# B&R Automation Studio project Pachore_Mayuresh_Project_1
Automation Studio 4.12.6.106; technology packages: Acp10Arnc0 5.24.1, mapp 5.24.1, mappView 5.24.4

## Configuration Config1

CPU X20CP1382, AutomationRuntime A4.83, Build 4.1.2, Safety 0.0, Vc V4.72.5

### Hardware
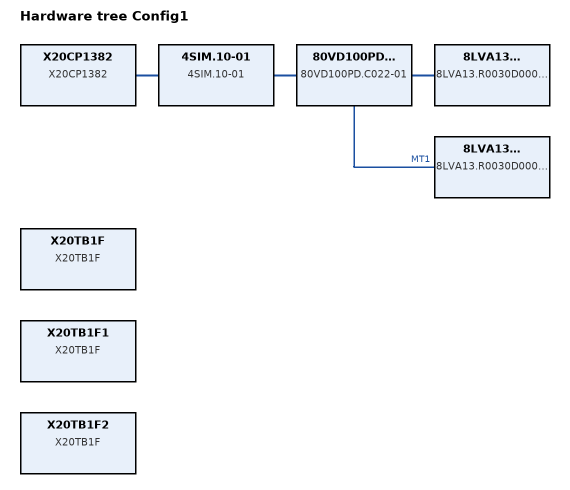
```
4SIM.10-01 : 4SIM.10-01 v1.3.0.0  [PLK1 -> X20CP1382.IF3 (NodeNumber=1) [Cable Type=PowerlinkCable, Length=10, Version=1.0.0.3]; PLK2 -> 80VD100PD.C022-01.PLK1 (NodeNumber=1) [Cable Type=PowerlinkCable, Length=10, Version=1.0.0.3]]
  Supervision = off
80VD100PD.C022-01 : 80VD100PD.C022-01 v2.5.0.0  [PLK1 -> 4SIM.10-01.PLK2 (NodeNumber=2) [Cable Type=PowerlinkCable, Length=10, Version=1.0.0.3]; MT2 -> 8LVA13.R0030D000-0.MT]
  MotionTP = Acp10Arnc0
  AxisIsPeriodic_r1 = on
  Period_r1 = 360
  BothEndSwitchesAreNormallyOpen_r1 = on
  QuickStopIsNormallyOpen_r1 = on
  AxisIsPeriodic_r2 = on
  Period_r2 = 360
  BothEndSwitchesAreNormallyOpen_r2 = on
  QuickStopIsNormallyOpen_r2 = on
8LVA13.R0030D000-0 : 8LVA13.R0030D000-0 v2.2.0.4  [MT -> 80VD100PD.C022-01.MT2]
8LVA13.R0030D000-0a : 8LVA13.R0030D000-0 v2.2.0.4  [MT -> 80VD100PD.C022-01.MT1]
X20CP1382 : X20CP1382 v1.14.0.0  [X1 -> X1.SL; X2 -> X2.SL; X3 -> X3.SL]
  Module X1 (Type=X1, Virtual=true, Version=1.14.0.0)
    Connection (Connector=SS1, TargetModule=X20TB1F, TargetConnector=SS)
    Connection (Connector=SL, TargetModule=X20CP1382, TargetConnector=X1)
  Module X2 (Type=X2, Virtual=true, Version=1.14.0.0)
    Connection (Connector=SS1, TargetModule=X20TB1F1, TargetConnector=SS)
    Connection (Connector=SL, TargetModule=X20CP1382, TargetConnector=X2)
  Module X3 (Type=X3, Virtual=true, Version=1.14.0.0)
    Connection (Connector=SS1, TargetModule=X20TB1F2, TargetConnector=SS)
    Connection (Connector=SL, TargetModule=X20CP1382, TargetConnector=X3)
  Connector IF2:
    ActivateDevice = 1
    Mode = Manual
    InternetAddress = 192.168.0.1
    SubnetMask = 255.255.255.0
    ActivateSnmp = 2
  Connector IF3:
    CycleTime = 2000
  ConfigurationID = UniboTest2024_Config1
  TimerDeviceType = EPLX2X
  TimerDevice = X20CP1382.IF3
  TaskClassIdleTime = 6000
  Cyclic1Duration = 2000
  Cyclic1Tolerance = 0
  ActivateOpcUa = 1
  OpcUaInformationModels_PV_Version = 1
X20TB1F : X20TB1F v1.0.0.0
X20TB1F1 : X20TB1F v1.0.0.0
X20TB1F2 : X20TB1F v1.0.0.0
```

### IoMap.iom - X20CP1382/IoMap.iom
```iecst
VAR_CONFIG
	::Conv_Lock AT %IX."4SIM.10-01".DigitalInput01;
	::Cutter_Lock AT %IX."4SIM.10-01".DigitalInput02;
	::Start_Button AT %IX."4SIM.10-01".DigitalInput03;
	::Stop_Button AT %IX."4SIM.10-01".DigitalInput04;
	::Sensor_Button AT %IX."4SIM.10-01".DigitalInput05;
	::Reset_Button AT %IX."4SIM.10-01".DigitalInput06;
	::Speed AT %IW."4SIM.10-01".AnalogInput01;
	::Position AT %IW."4SIM.10-01".AnalogInput02;
	::DI1.LED_Light AT %QX."4SIM.10-01".DigitalOutput01;
	::DI2.LED_Light AT %QX."4SIM.10-01".DigitalOutput02;
	::DI3.LED_Light AT %QX."4SIM.10-01".DigitalOutput05;
	::DI4.LED_Light AT %QX."4SIM.10-01".DigitalOutput06;
	::DI5.LED_Light AT %QX."4SIM.10-01".DigitalOutput10;
	::DI6.LED_Light AT %QX."4SIM.10-01".DigitalOutput12;
	::Display AT %QW."4SIM.10-01".AnalogOutput01;
END_VAR
```

### Acp10cfg.ncc - X20CP1382/Motion/Acp10cfg.ncc
```
NcConfiguration (Version=5.20.1, NcSwId=Acp10)
  ACP10CF1_typ:
    cnt_nettrc_rec_drive = 150
    bufsize_trace_upload = 1200
    tc_nc_man_task = Cyclic #1
    glob_pv_as_ncobject = Yes
    ncsys_dl_broadcast = Yes
    ncsys_dl_acp_reset = Yes
    safemc_log_err_to_ax = Yes
    network_init:
      ncsw_init_execute = Yes
      automatic_execute = No
      node_nr_warning = Yes
      net_err_before_ncact = Yes
    nettrc:
      enter_parsecrec = Yes
      enter_ncaction = Yes
      save_ring_startidx = No
    cam_prof_download:
      cam_dat_dl_parallel = No
      tc_cam_dl_parallel = Task class for NC Manager task
    plk_if[0]:
      if_name = IF3
      tc_CycDat_PLCopen = Task class for NC Manager task
      mc_broadcast_extdat = No
```

### Config.mpaxisbasic - X20CP1382/Motion/Config.mpaxisbasic
```
Element gAxisBasic_Master (Type=mpaxisbasic)
Element gAxisBasic_Slave (Type=mpaxisbasic)
```

## Logical view

Binary libraries used (declarations not repeated): operator, runtime, astime, AsIecCon, sys_lib, brsystem, Acp10man, Acp10par, NcGlobal, Acp10sim, Acp10_MC, MpAxis, AsTCP, standard, AsArLog, AsBrStr, MpBase, MpCom, AsIODiag

### MNG_Package.var
```iecst
(*                                                                            *)
(* File generated by the B&R AS 4 control config generator                    *)
(*                                                                            *)
(*     Provider: machineering                                                 *)
(*  Application: industrialPhysics_2.4.master                                 *)
(* Architecture: Windows 64 Bit                                               *)
(*      Version: 2.4.10491.master                                             *)
(*        Build: 164f85bec                                                    *)
(*         Date: 2020-03-30, Time: 13:49:25                                   *)
(*                                                                            *)

                VAR
                ComTCP_SimInputs : ComTCP_INPUTS_32BIT := (0);
    ComTCP_SimOutputs : ComTCP_OUTPUTS_32BIT := (0);

    ComTCP_SimServerAddress : STRING[15] := '127.0.0.1';
    ComTCP_SimServerPort : UINT := 5000;
    ComTCP_SimSendCycleTime : TIME := T#10ms;
    ComTCP_SimActive : BOOL := FALSE;

                END_VAR
```

### MNG_Package.typ
```iecst
(*                                                                            *)
(* File generated by the B&R AS 4 control config generator                    *)
(*                                                                            *)
(*     Provider: machineering                                                 *)
(*  Application: industrialPhysics_2.4.master                                 *)
(* Architecture: Windows 64 Bit                                               *)
(*      Version: 2.4.10491.master                                             *)
(*        Build: 164f85bec                                                    *)
(*         Date: 2020-03-30, Time: 13:49:25                                   *)
(*                                                                            *)

TYPE
ComTCP_INPUTS_32BIT : STRUCT

		NumSignals	: INT := 15;

        Emergency_Button_ButtonToggle : BOOL := 0;
        (* BOOL Emergency_Button_ButtonToggle *)
        Yellow_Button_ButtonPress : BOOL := 0;
        (* BOOL Yellow_Button_ButtonPress *)
        White_Button_ButtonPress : BOOL := 0;
        (* BOOL White_Button_ButtonPress *)
        Start_Button_ButtonPress : BOOL := 0;
        (* BOOL Start_Button_ButtonPress *)
        Stop_Button_ButtonPress : BOOL := 0;
        (* BOOL Stop_Button_ButtonPress *)
        Knob_0_AXIS : REAL := 0.0;
        (* REAL Knob_0_AXIS *)
        Knob_1_AXIS : REAL := 0.0;
        (* REAL Knob_1_AXIS *)
        Knob_2_AXIS : REAL := 0.0;
        (* REAL Knob_2_AXIS *)
        Knob_3_AXIS : REAL := 0.0;
        (* REAL Knob_3_AXIS *)
        Shaft_1_AXIS : REAL := 0.0;
        (* REAL Shaft_1_AXIS *)
        Shaft_1_LBK : BOOL := 0;
        (* BOOL Shaft_1_LBK *)
        Shaft_1_LFR : BOOL := 0;
        (* BOOL Shaft_1_LFR *)
        Shaft_0_AXIS : REAL := 0.0;
        (* REAL Shaft_0_AXIS *)
        Shaft_0_LBK : BOOL := 0;
        (* BOOL Shaft_0_LBK *)
        Shaft_0_LFR : BOOL := 0;
        (* BOOL Shaft_0_LFR *)

	END_STRUCT;

ComTCP_OUTPUTS_32BIT : STRUCT

		NumSignals	: INT := 6;

        Yellow_light_Key : UDINT := 0;
        (* UDINT Yellow_light_Key *)
        Stop_light_Key : UDINT := 0;
        (* UDINT Stop_light_Key *)
        White_light_Key : UDINT := 0;
        (* UDINT White_light_Key *)
        Green_light_Key : UDINT := 0;
        (* UDINT Green_light_Key *)
        Shaft_0_ACT_POS : REAL := 0.0;
        (* REAL Shaft_0_ACT_POS *)
        Shaft_1_ACT_POS : REAL := 0.0;
        (* REAL Shaft_1_ACT_POS *)

	END_STRUCT;

END_TYPE
```

### Global.var - Global variables
```iecst
(*Name of Axis*)
VAR
	gAxis01 : ACP10AXIS_typ;
	gAxis02 : ACP10AXIS_typ;
END_VAR
(*Hardware Variables*)
VAR
	Conv_Lock : BOOL;
	Cutter_Lock : BOOL;
	Start_Button : BOOL;
	Stop_Button : BOOL;
	Sensor_Button : BOOL;
	Reset_Button : BOOL;
	Speed : INT;
	Position : INT;
	DI1 : FSM_LED;
	DI2 : FSM_LED;
	DI3 : FSM_LED;
	DI4 : FSM_LED;
	DI5 : FSM_LED;
	DI6 : FSM_LED;
	Display : INT;
END_VAR
(*HMI Variables*)
VAR
	Emergancy_Button_HMI : BOOL;
	Start_Button_HMI : BOOL;
	Stop_Button_HMI : BOOL;
	Sensor_Button_HMI : BOOL;
	Reset_Button_HMI : BOOL;
	Conv_Lock_HMI : BOOL;
	Cutter_Lock_HMI : BOOL;
	Conv_Speed_HMI : REAL;
	Cutter_Speed_HMI : REAL;
	Cutting_Pos_HMI : REAL;
	Cutting_Depth_HMI : REAL;
	Blade_Man_HMI : REAL;
	Conv_Man_HMI : REAL;
	Slow_Blade_HMI : BOOL;
	Slow_Conv_HMI : BOOL;
	LED_DI1_HMI : BOOL;
	LED_DI2_HMI : BOOL;
	LED_DI3_HMI : BOOL;
	LED_DI4_HMI : BOOL;
	LED_DI5_HMI : BOOL;
	LED_DI6_HMI : BOOL;
	Dis_Conv_Speed_HMI : REAL;
	Dis_Cut_Speed_HMI : REAL;
	Dis_Cut_Pos_HMI : INT;
	Dis_Cut_Depth_HMI : INT;
	Man_Mode_HMI : BOOL;
	Over_Ride_HMI : BOOL;
END_VAR
(*LED_IO Variables*)
VAR
	Power_Axis : BOOL;
	Home_Axis : BOOL;
	Reset_Command : BOOL;
	Error_Command : BOOL;
	Start_Command : BOOL := FALSE;
	Stop_Command : BOOL := TRUE;
END_VAR
(*Master Variables*)
VAR
	Master : FSM_AXIS;
	M_Active : BOOL;
	M_Actual_Position : REAL;
	M_Actual_Velocity : REAL;
	M_Homed : BOOL;
	M_Powered : BOOL;
	M_Stoped : BOOL;
	Do_Cut : BOOL := FALSE;
	Done_Cut : BOOL := FALSE;
END_VAR
(*Slave Variables*)
VAR
	Slave : FSM_AXIS;
	S_Active : BOOL;
	S_Actual_Position : REAL;
	S_Actual_Velocity : REAL;
	S_Homed : BOOL;
	S_Powered : BOOL;
	S_Stoped : BOOL;
END_VAR
(*Input Bridge Variables*)
VAR
	Start_Trigger : BOOL;
	Stop_Trigger : BOOL;
	Error_Trigger : BOOL;
	Reset_Trigger : BOOL;
	Sensor_Trigger : BOOL;
	Conv_Lock_HMI_Trigger : BOOL;
	Conv_Lock_Trigger : BOOL;
	Cutter_Lock_HMI_Trigger : BOOL;
	Cutter_Lock_Trigger : BOOL;
	Slow_Blade_Trigger : BOOL;
	Slow_Conv_Trigger : BOOL;
	Over_Ride_Trigger : BOOL;
	Conv_Speed : REAL;
	Cut_Pos : REAL;
	Cutter_Speed : REAL;
	Cut_depth : REAL;
	Blade_Pos : REAL;
	Conv_Pos : REAL;
	M_Error : BOOL;
	S_Error : BOOL;
END_VAR
(*Manual Motion Variables*)
VAR
	Manual_Mode_Trigger : BOOL;
	Man_Mode_OFF : BOOL := TRUE;
END_VAR
```

### Package Logical/Libraries - Global libraries

### Library Logical/Libraries/ComTCP/ComTCP_L (ANSIC)

#### MNG_ComHdlr.cpp
```cpp
#include "MNG_ComHdlr.hpp"
#include "MNG_CpyMsgToInp.cpp"
#include "MNG_CpyOutToMsg.cpp"

asTcpFcn_t _asTcpFcn;

MNG_ComHdlr::MNG_ComHdlr(char *srvIpAdr, unsigned int srvPort, TIME sendCycleTime)
{
	_srvIpAdr = srvIpAdr;
	_srvPort = srvPort;
	_sendCycleTime = sendCycleTime;
	InitParams();
}

MNG_ComHdlr::~MNG_ComHdlr()
{
}

int MNG_ComHdlr::RunCommunication(void* pSimInputs, void* pSimOutputs, BOOL* pSimActive) {

        unsigned long int _lastCounter = _counter;

	ComTCP_INPUTS_32BIT_FWRD* pFwrd_SimInputs = static_cast<ComTCP_INPUTS_32BIT_FWRD*>((pSimInputs));
	ComTCP_OUTPUTS_32BIT_FWRD* pFwrd_SimOutputs = static_cast<ComTCP_OUTPUTS_32BIT_FWRD*>((pSimOutputs));

	switch (_internalState) {

		case MNG_Init:
                        *pSimActive = FALSE;
			_asTcpFcn.tcpOpen.enable = FALSE;
			TcpOpen(&_asTcpFcn.tcpOpen);
			_asTcpFcn.tcpIoctl.enable = FALSE;
			TcpIoctl(&_asTcpFcn.tcpIoctl);
			_asTcpFcn.tcpClient.enable = FALSE;
			TcpClient(&_asTcpFcn.tcpClient);
			_asTcpFcn.tcpSend.enable = FALSE;
			TcpSend(&_asTcpFcn.tcpSend);
			_asTcpFcn.tcpRecv.enable = FALSE;
			TcpRecv(&_asTcpFcn.tcpRecv);
			_asTcpFcn.tcpClose.enable = FALSE;
			TcpClose(&_asTcpFcn.tcpClose);

			_connectionTon.IN = FALSE;
			_connectionTon.PT = _connectionTime;
			_sendTon.IN = FALSE;
			_sendTon.PT = _sendCycleTime;
			SetStateValue(MNG_Socket);
			break;

		case MNG_Socket:
                        *pSimActive = FALSE;
			init_TcpSocket();
			TcpOpen(&_asTcpFcn.tcpOpen);
			_recvOffset = 0;
			if (_connect == 1) {
				SetStateValue(MNG_Open);
				_connectionTon.IN = FALSE;
			}
			break;

		case MNG_Open:
                        *pSimActive = FALSE;
			init_TcpOpen();
			TcpOpen(&_asTcpFcn.tcpOpen);
			if (_asTcpFcn.tcpOpen.status == 0) {
				SetStateValue(MNG_SetIo);
				_asTcpFcn.tcpIoctl.enable = FALSE;
				TcpIoctl(&_asTcpFcn.tcpIoctl);
				_connectionTon.IN = FALSE;
			}
			break;

		case MNG_SetIo:
                        *pSimActive = FALSE;
			init_TcpIoctl();
			TcpIoctl(&_asTcpFcn.tcpIoctl);
			if (_asTcpFcn.tcpIoctl.status == 0) {
				SetStateValue(MNG_Linger);
				_asTcpFcn.tcpClient.enable = FALSE;
				TcpClient(&_asTcpFcn.tcpClient);
				_connectionTon.IN = FALSE;
			}
			break;

		case MNG_Linger:
                        *pSimActive = FALSE;
			init_TcpLinger();
			TcpIoctl(&_asTcpFcn.tcpIoctl);

			if (_asTcpFcn.tcpIoctl.status == 0) {
				SetStateValue(MNG_Connecting);
				_asTcpFcn.tcpClient.enable = FALSE;
				_connectionTon.IN = FALSE;
			}

		case MNG_Connecting:
                        *pSimActive = FALSE;
			_asTcpFcn.tcpClient.enable = TRUE;
			_asTcpFcn.tcpClient.ident = _asTcpFcn.tcpOpen.ident;
			_asTcpFcn.tcpClient.portserv = _srvPort;
			_asTcpFcn.tcpClient.pServer = (long)_srvIpAdr;
			TcpClient(&_asTcpFcn.tcpClient);

			if (_asTcpFcn.tcpClient.status == ERR_FUB_BUSY) {
				// state = state || SetStateValue(Connecting);
			} else if (_asTcpFcn.tcpClient.status == 0) {
				SetStateValue(MNG_Exchange);
				_connectionTon.IN = FALSE;
				SetSendDone(TRUE);
			}
			break;

		case MNG_Exchange:
			init_TcpRecv();
			TcpRecv(&_asTcpFcn.tcpRecv);

			if (_asTcpFcn.tcpRecv.status==0){
                        *pSimActive = FALSE;
			_connectionTon.IN = FALSE;
			_recvLen = _asTcpFcn.tcpRecv.recvlen;
			_potMsgLen = N_TO_HUDINT(_recvBuffer[3]) + SIXTEEN;
			_totalRecvLen = _recvOffset + _recvLen;

			if ((_totalRecvLen < SIXTEEN) || (_totalRecvLen < _potMsgLen)) {
			_recvOffset = _recvOffset + _recvLen;
			}	else {
			while ((_potMsgLen > 0) && (_potMsgLen <= _totalRecvLen)) {
			// misconfigured message sizes
                        if ((unsigned long int)_potMsgLen > sizeof(_recvMessage)) {
			SetStateValue(MNG_Reset);
			break;
			}

			brsmemcpy((unsigned long int) &_recvMessage, (unsigned long int) &_recvBuffer, _potMsgLen*sizeof(unsigned long int));
			_totalRecvLen = _totalRecvLen - _potMsgLen;
			brsmemmove((unsigned long int) &_recvBuffer, (unsigned long int) &_recvBuffer + _potMsgLen, _totalRecvLen*sizeof(unsigned long int));
			_counter = MNG_CpyMsgToInp(&_recvMessage,pFwrd_SimInputs);
                        *pSimActive = (_lastCounter != _counter);
			_recvOffset = _totalRecvLen;

			if (_totalRecvLen > SIXTEEN) {
			_potMsgLen = N_TO_HUDINT(_recvBuffer[3]) + SIXTEEN;
			} else {
			_potMsgLen = 0;
			}

			}
			}
			}

			_sendTon.IN = _sendDone;
			TON(&_sendTon);

			if (_sendTon.Q || _asTcpFcn.tcpSend.enable == 1) {
				if (_sendDone==TRUE) {
					SetSendDone(FALSE);
					MNG_CpyOutToMsg(&_sendMessage, _counter,pFwrd_SimOutputs);
					init_TcpSend(pFwrd_SimOutputs);
				}
				TcpSend(&_asTcpFcn.tcpSend);

				if (_asTcpFcn.tcpSend.status == 0) {
					if (_asTcpFcn.tcpSend.datalen != _asTcpFcn.tcpSend.sentlen) {
						// state = state || SetStateValue(Exchange);
					}
					_asTcpFcn.tcpSend.enable = FALSE;
					SetSendDone(TRUE);
				}
			}
			if (_asTcpFcn.tcpRecv.status == tcpERR_NOT_CONNECTED) {
				SetStateValue(MNG_Closing);
			}
			break;

		case MNG_Closing:
                        *pSimActive = FALSE;
			_asTcpFcn.tcpClose.enable = TRUE;
			_asTcpFcn.tcpClose.ident = _asTcpFcn.tcpOpen.ident;
			_asTcpFcn.tcpClose.how = 0;
			TcpClose(&_asTcpFcn.tcpClose);

			if(_asTcpFcn.tcpClose.status == 0 || _asTcpFcn.tcpClose.status == 32600){
				SetStateValue(MNG_Init);
			}
			break;

                case MNG_Reset:
                        SetStateValue(MNG_Closing);
                        break;
	}

	TON(&_connectionTon);
	_connectionTon.IN = TRUE;
	if (_connectionTon.Q == 1) {
		SetStateValue(MNG_Closing);
		_connectionTon.IN = FALSE;
	}

	return _internalState;
}

void MNG_ComHdlr::init_TcpOpen(){
	_asTcpFcn.tcpOpen.enable = _connect;
}

void MNG_ComHdlr::init_TcpSocket(){
	_asTcpFcn.tcpOpen.enable = TRUE;
	_asTcpFcn.tcpOpen.pIfAddr = 0;
	_asTcpFcn.tcpOpen.port = PORT;
	_asTcpFcn.tcpOpen.options = tcpOPT_REUSEADDR;
}

void MNG_ComHdlr::init_TcpIoctl(){
	_asTcpFcn.tcpIoctl.enable = TRUE;
	_asTcpFcn.tcpIoctl.pData = (unsigned long int) &_one;
	_asTcpFcn.tcpIoctl.datalen = 4;
	_asTcpFcn.tcpIoctl.ident = _asTcpFcn.tcpOpen.ident;
	_asTcpFcn.tcpIoctl.ioctl = tcpTCP_NODELAY_SET;
}

void MNG_ComHdlr::init_TcpLinger(){
	_asTcpFcn.tcpLINGER.lLinger = FALSE;
	_asTcpFcn.tcpLINGER.lOnOff = TRUE;
	_asTcpFcn.tcpIoctl.enable = TRUE;
	_asTcpFcn.tcpIoctl.pData = (unsigned long int) &_asTcpFcn.tcpLINGER;
	_asTcpFcn.tcpIoctl.datalen = sizeof(_asTcpFcn.tcpLINGER);
	_asTcpFcn.tcpIoctl.ident = _asTcpFcn.tcpOpen.ident;
	_asTcpFcn.tcpIoctl.ioctl = tcpSO_LINGER_SET;
}

void MNG_ComHdlr::init_TcpClient(){

	_asTcpFcn.tcpClient.enable = TRUE;
	_asTcpFcn.tcpClient.ident = _asTcpFcn.tcpOpen.ident;
	_asTcpFcn.tcpClient.portserv = _srvPort;
	_asTcpFcn.tcpClient.pServer = (long)_srvIpAdr;
}

void MNG_ComHdlr::init_TcpRecv(){

	_asTcpFcn.tcpRecv.enable = TRUE;
	_asTcpFcn.tcpRecv.ident= _asTcpFcn.tcpOpen.ident;
	_asTcpFcn.tcpRecv.datamax = sizeof(_recvBuffer) - _recvOffset;
	_asTcpFcn.tcpRecv.pData = (unsigned long int) &_recvBuffer + _recvOffset;
}

void MNG_ComHdlr::init_TcpSend(ComTCP_OUTPUTS_32BIT_FWRD *pSimOutputs){

	_asTcpFcn.tcpSend.enable = TRUE;
	_asTcpFcn.tcpSend.ident= _asTcpFcn.tcpOpen.ident;
	_asTcpFcn.tcpSend.datalen = 16 + ((pSimOutputs->NumSignals) + 1) * 4;
	_asTcpFcn.tcpSend.pData = (unsigned long int)&_sendMessage;
	_asTcpFcn.tcpSend.flags = 0;
}

void MNG_ComHdlr::InitParams(){
	_internalState = MNG_Init;
	_connectionTime = 3000;
	_one=1;
	_connect = TRUE;
	_potMsgLen = 0;
	_recvLen = 0;
	_recvOffset = 0;
	_counter = 0;
	SetSendDone(FALSE);
}

void MNG_ComHdlr::SetSendDone(bool toggle){
	_sendDone=toggle;
}

void MNG_ComHdlr::SetStateValue(MNG_internalState_t stateVal){
	_internalState=stateVal;
}
```

#### MNG_CpyOutToMsg.cpp
```cpp
#include "MNG_InternalTyp.hpp"

unsigned long int MNG_CpyOutToMsg(MNG_RawDatagram * pToServer, unsigned long int counter, ComTCP_OUTPUTS_32BIT_FWRD *pSimOutputs ) {

        unsigned long int DWordBuffer;

        pSimOutputs->NumSignals = 6;
        (pToServer->Header).ByteCount    = H_TO_NUDINT(28);
        (pToServer->Header).DatagramType = H_TO_NUDINT(MNG_Raw32BitImage);
        (pToServer->Header).SentTime = H_TO_NUDINT(0);  // Todo
        (pToServer->Header).Counter = H_TO_NUDINT(counter);
        pToServer->Payload[0] = H_TO_NUDINT(pSimOutputs->NumSignals);

    /* Yellow_light_Key : UINT32 */
    pToServer->Payload[1] = H_TO_NUDINT(pSimOutputs->Yellow_light_Key);

    /* Stop_light_Key : UINT32 */
    pToServer->Payload[2] = H_TO_NUDINT(pSimOutputs->Stop_light_Key);

    /* White_light_Key : UINT32 */
    pToServer->Payload[3] = H_TO_NUDINT(pSimOutputs->White_light_Key);

    /* Green_light_Key : UINT32 */
    pToServer->Payload[4] = H_TO_NUDINT(pSimOutputs->Green_light_Key);

    /* Shaft_0_ACT_POS : FLOAT32 */
    brsmemcpy((unsigned long int)&(DWordBuffer), (unsigned long int)&(pSimOutputs->Shaft_0_ACT_POS), 4);
    pToServer->Payload[5] = H_TO_NUDINT(DWordBuffer);

    /* Shaft_1_ACT_POS : FLOAT32 */
    brsmemcpy((unsigned long int)&(DWordBuffer), (unsigned long int)&(pSimOutputs->Shaft_1_ACT_POS), 4);
    pToServer->Payload[6] = H_TO_NUDINT(DWordBuffer);

	return 0;
}
```

### Library Logical/Libraries/My_Library (IEC)

#### FSM_AXIS.st
```iecst
FUNCTION_BLOCK FSM_AXIS

	CASE State OF
		0://Initiation
			Power_ON := FALSE;

			IF RS_Valid AND RS_Disabled THEN
				State 	:= 2;
				Active 	:= TRUE;
			END_IF

			IF RS_Errorstop AND RS_Valid THEN
				State 	:= 1;
			END_IF

		1://Error
			V_Execute 	:= FALSE;
			Add_Execute := FALSE;
			A_Execute 	:= FALSE;

			IF Reset_Error THEN
				R_Execute := TRUE;
				IF R_Done AND P_Status THEN
					State := 3;
				END_IF
				IF R_Done AND NOT P_Status THEN
					State := 2;
				END_IF
			END_IF

		2://Disabled
			P_Enable := FALSE;
			Power_ON := FALSE;

			IF Error THEN
				State := 1;
			ELSIF Home THEN
				State := 4;
			ELSIF Power THEN
				State := 3;
			END_IF

		3://StandStill

			P_Enable := TRUE;
			Power_ON := TRUE;

			IF Error THEN
				State 			:= 1;
			ELSIF Home AND NOT Is_Homed THEN
				State 			:= 4;
			ELSIF NOT Power THEN
				State 			:= 2;
			ELSIF Move_Velocity THEN
				Move_Abs_Done 	:= FALSE;
				Move_Add_Done 	:= FALSE;
				Stop_Done 		:= FALSE;
				State 			:= 5;
			ELSIF Move_Additive AND NOT Move_Additive_Old THEN
				Move_Abs_Done 	:= FALSE;
				Move_Add_Done 	:= FALSE;
				Stop_Done 		:= FALSE;
				State 			:= 6;
			ELSIF Move_Absolute AND NOT Move_Absolute_Old THEN
				Move_Abs_Done 	:= FALSE;
				Move_Add_Done 	:= FALSE;
				Stop_Done 		:= FALSE;
				State 			:= 7;
			ELSIF Stop THEN
				State 			:= 8;
			END_IF

		4://Homing Axis

			H_Execute := TRUE;
			IF Error THEN
				State 		:= 1;
				H_Execute 	:= FALSE;
			ELSIF H_Done AND Power THEN
				State 		:= 3;
				H_Execute 	:= FALSE;
				Is_Homed 	:= TRUE;
			ELSIF H_Done AND NOT Power THEN
				State 		:= 2;
				H_Execute 	:= FALSE;
				Is_Homed 	:= TRUE;
			END_IF

		5://Moving Axis in Velocity mode

			P_Enable 	:= TRUE;
			V_Execute 	:= TRUE;
			IF Old_Velocity <> Velocity THEN
				V_Execute := FALSE;
			END_IF

			IF Error THEN
				State := 1;
			ELSIF Move_Additive THEN
				State := 6;
			ELSIF Move_Absolute THEN
				State := 7;
			ELSIF NOT Power OR Stop THEN
				State := 8;
			END_IF

		6://Moving Axis in Additive mode

			P_Enable 	:= TRUE;
			Add_Execute := TRUE;

			IF Error THEN
				State 			:= 1;
			END_IF
			IF NOT Power OR Stop THEN
				State 			:= 8;
				Add_Execute 	:= FALSE;
			END_IF
			IF Add_Done THEN
				Move_Add_Done 	:= TRUE;
				Add_Execute 	:= FALSE;
				State 			:= 3;
			END_IF

		7://Moving Axis in Absolute Mode

			P_Enable 	:= TRUE;
			A_Execute 	:= TRUE;

			IF Error THEN
				State 			:= 1;
			END_IF
			IF NOT Power OR Stop THEN
				State 			:= 8;
				A_Execute 		:= FALSE;
			END_IF
			IF A_Done THEN
				Move_Abs_Done 	:= TRUE;
				A_Execute 		:= FALSE;
				State 			:= 3;
			END_IF

		8://Stopping Axis

			P_Enable 	:= TRUE;
			S_Execute 	:= TRUE;

			IF Error THEN
				State 		:= 1;
			END_IF
			IF S_Done THEN
				V_Execute 	:= FALSE;
				S_Execute 	:= FALSE;
				Stop_Done 	:= TRUE;
				State 		:= 3;
			END_IF
			IF RS_Errorstop AND RS_Valid THEN
				S_Execute 	:= FALSE;
				State 		:= 1;
			END_IF

	END_CASE

	Move_Absolute_Old 		:= Move_Absolute;
	Move_Additive_Old 		:= Move_Additive;
	Old_Velocity 			:= Velocity;

	//Calling all PLCopen function blocks used
	//Read Status
	MCRS(	Axis 			:= Axis_Name,
			Enable 			:= TRUE);
	RS_Valid 				:= MCRS.Valid;
	RS_Error 				:= MCRS.Error;
	RS_Errorstop 			:= MCRS.Errorstop;
	RS_Disabled 			:= MCRS.Disabled;
	//Power
	MCP(	Axis 			:= Axis_Name,
			Enable 			:= P_Enable);
	P_Status 				:= MCP.Status;
	P_Error 				:= MCP.Error;
	//Home
	MCH(	Axis 			:= Axis_Name,
			Execute 		:= H_Execute);
	H_Done 					:= MCH.Done;
	H_Error					:= MCH.Error;
	//Stop
	MCS(	Axis 			:= Axis_Name,
			Execute 		:= S_Execute,
			Deceleration 	:= Deceleration);
	S_Done 					:= MCS.Done;
	S_Error 				:= MCS.Error;
	//Reset
	MCR(	Axis 			:= Axis_Name,
			Execute			:= R_Execute);
	R_Done 					:= MCR.Done;
	R_Error 				:= MCR.Error;
	//Read Actual Position
	MCRAP(	Axis 			:= Axis_Name,
			Enable 			:= TRUE);
	RAP_Valid 				:= MCRAP.Valid;
	RAP_Error 				:= MCRAP.Error;
	Actual_Position 		:= MCRAP.Position;
	//Read Actual Velocity
	MCRAV(	Axis 			:= Axis_Name,
			Enable 			:= TRUE);
	RAV_Valid 				:= MCRAV.Valid;
	RAV_Error 				:= MCRAV.Error;
	Actual_Velocity 		:= MCRAV.Velocity;
	//Move Velocity
	MCMV(	Axis 			:= Axis_Name,
			Execute 		:= V_Execute,
			Velocity 		:= Velocity,
			Acceleration 	:= Acceleration,
			Deceleration 	:= Deceleration,
			Direction 		:= Direction);
	V_Error 				:= MCMV.Error;
	//Move Additive
	MCMAdd(	Axis 			:= Axis_Name,
			Execute 		:= Add_Execute,
			Distance 		:= Distance,
			Velocity 		:= Velocity,
			Acceleration 	:= Acceleration,
			Deceleration 	:= Deceleration);
	Add_Done 				:= MCMAdd.Done;
	Add_Error 				:= MCMAdd.Error;
	//Move Absolute
	MCMA(	Axis 			:= Axis_Name,
			Execute 		:= A_Execute,
			Position 		:= Position,
			Velocity 		:= Velocity,
			Acceleration 	:= Acceleration,
			Deceleration 	:= Deceleration,
			Direction 		:= Direction);
	A_Done 					:= MCMA.Done;
	A_Error 				:= MCMA.Error;

	Error := RS_Error OR P_Error OR H_Error OR S_Error OR R_Error OR RAP_Error OR RAV_Error OR V_Error OR Add_Error OR A_Error;

END_FUNCTION_BLOCK
```

#### FSM_LED.st
```iecst
(* For Turning LED ON/OFF/Blink *)
FUNCTION_BLOCK FSM_LED

	IF LED_State = 'on' THEN
		LED_Light := TRUE;
	END_IF

	IF LED_State = 'off' THEN
		LED_Light := FALSE;
	END_IF

	IF LED_State = 'blink' THEN

		CASE State OF

			0:
				Timer(IN := TRUE, PT := T#500ms);
				IF Timer.Q = TRUE THEN
					Timer(IN 	:= FALSE);
					LED_Light 	:= TRUE;
					State 		:= 1;
				END_IF

			1:
				Timer(IN := TRUE, PT := T#500ms);
				IF Timer.Q = TRUE THEN
					Timer(IN 	:= FALSE);
					LED_Light 	:= FALSE;
					State 		:= 0;
				END_IF
		END_CASE

	END_IF

END_FUNCTION_BLOCK
```


- Data object Logical/gAxis01obj/gAxis01i (Ax) (no source held here)

- Data object Logical/gAxis02obj/gAxis02i (Ax) (no source held here)

### Data object Logical/MyCam (Cam)

- Visualisation Logical/mappView (not shown)

### Program Logical/Master (IEC)

#### Variables.var
```iecst
VAR
	M_Move_Velocity : BOOL;
	M_Move_Additive : BOOL;
	M_Move_Absolute : BOOL;
	M_Stop : BOOL;
	State : INT := 0;
	M_Position : REAL;
	one_time : BOOL;
	M_Move_Additive_Done : BOOL;
	M_Move_Absolute_Done : BOOL;
	M_Distance : REAL;
	M_Direction : USINT := 0;
	M_Velocity : REAL;
END_VAR
```

#### Main.st
```iecst
PROGRAM _INIT
	(* Insert code here *)

END_PROGRAM

PROGRAM _CYCLIC

	CASE State OF
		0://Initialization

			IF M_Active AND M_Homed AND M_Powered THEN
				State := 2;
			END_IF
			IF Manual_Mode_Trigger THEN
				State := 5;
			END_IF

		1://Error and Stopping

			M_Move_Velocity := FALSE;
			M_Move_Additive := FALSE;
			M_Move_Absolute := FALSE;
			M_Stop 			:= TRUE;

			IF M_Stoped THEN
				M_Move_Velocity := FALSE;
				M_Move_Additive := FALSE;
				M_Move_Absolute := FALSE;
				M_Stop 			:= FALSE;
				State 			:= 2;
			END_IF

		2://Standstill

			IF NOT Error_Command AND Start_Command AND Man_Mode_OFF AND (NOT Do_Cut OR Done_Cut) THEN
				State := 3;
			END_IF
			IF Manual_Mode_Trigger THEN
				State := 5;
			END_IF

		3://Moving Conveyor
			M_Velocity 		:= Conv_Speed;
			M_Move_Velocity := TRUE;
			M_Move_Additive := FALSE;
			M_Move_Absolute := FALSE;
			M_Stop 			:= FALSE;

			Do_Cut 		:= FALSE;
			Done_Cut 	:= FALSE;

			IF Stop_Command OR Error_Command THEN
				State := 1;
			ELSIF Sensor_Trigger THEN
				State := 4;
			ELSIF Manual_Mode_Trigger THEN
				State := 5;
			END_IF

		4://Reaching Cutting Position
			M_Distance 		:= Cut_Pos;
			M_Velocity 		:= Conv_Speed;
			M_Move_Velocity := FALSE;
			M_Move_Additive := TRUE;
			M_Move_Absolute := FALSE;
			M_Stop 			:= FALSE;

			IF M_Move_Additive_Done THEN
				State 			:= 1;
				Do_Cut 			:= TRUE;
				M_Move_Velocity := FALSE;
				M_Move_Additive := FALSE;
				M_Move_Absolute := FALSE;
				M_Stop 			:= FALSE;
				one_time 		:= FALSE;
			END_IF

			IF Stop_Command OR Error_Command THEN
				State := 1;
			END_IF

			IF Done_Cut AND NOT (Stop_Command OR Error_Command) THEN
				State := 2;
			END_IF

			IF Manual_Mode_Trigger THEN
				State := 5;
			END_IF

		5://Running in Manual Mode
			Power_Axis 		:= TRUE;
			Man_Mode_OFF 	:= FALSE;
			M_Move_Velocity := TRUE;
			M_Move_Additive := FALSE;
			M_Move_Absolute := FALSE;
			M_Stop 			:= FALSE;

			M_Velocity 		:= Conv_Pos;
			M_Direction 	:= 0;
			IF M_Velocity < 0 THEN
				M_Velocity 	:= -Conv_Pos;
				M_Direction := 1;
			END_IF
			IF NOT Manual_Mode_Trigger THEN
				Power_Axis 		:= FALSE;
				Start_Command 	:= FALSE;
				M_Move_Velocity := FALSE;
				M_Move_Additive := FALSE;
				M_Move_Absolute := FALSE;
				M_Stop 			:= FALSE;
				State 			:= 2;
			END_IF

			IF Error_Command THEN
				State := 1;
			END_IF

	END_CASE

	//Calling FSM_AXIS Function
	Master(	Axis_Name 		:= ADR(gAxis01),
			Acceleration 	:= 5000,
			Deceleration 	:= 5000,
			Position 		:= M_Position,
			Distance 		:= M_Distance,
			Velocity 		:= M_Velocity,
			Direction 		:= M_Direction,
			Home 			:= Home_Axis,
			Power 			:= Power_Axis,
			Move_Velocity 	:= M_Move_Velocity,
			Move_Absolute 	:= M_Move_Absolute,
			Move_Additive 	:= M_Move_Additive,
			Stop 			:= M_Stop,
			Reset_Error 	:= Reset_Command);
	M_Active 				:= Master.Active;
	M_Actual_Position		:= Master.Actual_Position;
	M_Actual_Velocity 		:= Master.Actual_Velocity;
	M_Move_Absolute_Done 	:= Master.Move_Abs_Done;
	M_Move_Additive_Done 	:= Master.Move_Add_Done;
	M_Homed 				:= Master.Is_Homed;
	M_Powered 				:= Master.Power_ON;
	M_Stoped 				:= Master.Stop_Done;
	M_Error 				:= Master.Error;

END_PROGRAM

PROGRAM _EXIT
	(* Insert code here *)

END_PROGRAM
```

### Program Logical/Slave (IEC)

#### Variables.var
```iecst
VAR
	State : INT := 0;
	S_Move_Velocity : BOOL;
	S_Move_Absolute : BOOL;
	S_Move_Additive : BOOL;
	S_Stop : BOOL;
	S_Move_Absolute_Done : BOOL;
	S_Direction : USINT;
	S_Move_Additive_Done : BOOL;
	S_Position : REAL;
	S_Distance : REAL;
	S_Velocity : REAL;
END_VAR
```

#### Main.st
```iecst
PROGRAM _INIT
	(* Insert code here *)

END_PROGRAM

PROGRAM _CYCLIC

	CASE State OF
		0://Initiation

			Done_Cut 	:= FALSE;
			Do_Cut 		:= FALSE;
			State 		:= 1;

		1://Standstill

			IF NOT Error_Command AND Start_Command AND Do_Cut AND Man_Mode_OFF THEN
				S_Velocity 	:= Cutter_Speed;
				State 		:= 2;     //Uncomment for Cutter in Cam similar Mechanism
				//State 		:= 4;   //Uncomment for Cutter in Lead Screw Mechanism
			END_IF

			IF Manual_Mode_Trigger THEN
				State := 6;
			END_IF

		2://Cutting Considering it as a Cam cutter
			S_Move_Velocity := FALSE;
			S_Move_Absolute := TRUE;
			S_Move_Additive := FALSE;
			S_Stop 			:= FALSE;
			S_Position 		:= Cut_depth;
			S_Direction 	:= 0;

			IF S_Actual_Position = 0.0 THEN
				S_Move_Absolute_Done := FALSE;
			END_IF

			IF S_Move_Absolute_Done THEN
				State 			:= 3;
				S_Move_Velocity := FALSE;
				S_Move_Absolute := FALSE;
				S_Move_Additive := FALSE;
				S_Stop 			:= FALSE;
			END_IF

			IF Stop_Command OR Error_Command OR NOT Do_Cut THEN
				State 			:= 1;
				S_Move_Velocity := FALSE;
				S_Move_Absolute := FALSE;
				S_Move_Additive := FALSE;
				S_Stop 			:= FALSE;
			END_IF

		3://Retracting Considering it as a Cam cutter
			S_Move_Velocity := FALSE;
			S_Move_Absolute := TRUE;
			S_Move_Additive := FALSE;
			S_Stop 			:= FALSE;
			S_Position 		:= 0.0;
			S_Direction 	:= 1;

			IF S_Actual_Position <> 0.0 THEN
				S_Move_Absolute_Done := FALSE;
			END_IF

			IF S_Move_Absolute_Done THEN
				State 			:= 1;
				Do_Cut 			:= FALSE;
				Done_Cut 		:= TRUE;
				S_Move_Velocity := FALSE;
				S_Move_Absolute := FALSE;
				S_Move_Additive := FALSE;
				S_Stop 			:= FALSE;
			END_IF

			IF Stop_Command OR Error_Command OR NOT Do_Cut THEN
				State 			:= 1;
				S_Move_Velocity := FALSE;
				S_Move_Absolute := FALSE;
				S_Move_Additive := FALSE;
				S_Stop 			:= FALSE;
			END_IF

		4://Cutting Considering a lead Screw Cutter
			S_Move_Velocity := FALSE;
			S_Move_Absolute := FALSE;
			S_Move_Additive := TRUE;
			S_Stop 			:= FALSE;
			S_Distance 		:= Cut_depth;

			IF S_Actual_Position = 0.0 THEN
				S_Move_Additive_Done := FALSE;
			END_IF

			IF S_Move_Additive_Done THEN
				State 			:= 5;
				S_Move_Velocity := FALSE;
				S_Move_Absolute := FALSE;
				S_Move_Additive := FALSE;
				S_Stop 			:= FALSE;
			END_IF

			IF Stop_Command OR Error_Command OR NOT Do_Cut THEN
				State 			:= 1;
				S_Move_Velocity := FALSE;
				S_Move_Absolute := FALSE;
				S_Move_Additive := FALSE;
				S_Stop 			:= FALSE;
			END_IF

		5://Retracting Considering a lead Screw Cutter
			S_Move_Velocity := FALSE;
			S_Move_Absolute := FALSE;
			S_Move_Additive := TRUE;
			S_Stop 			:= FALSE;
			S_Distance 		:= -Cut_depth;

			IF S_Actual_Position <> 0.0 THEN
				S_Move_Additive_Done := FALSE;
			END_IF

			IF S_Move_Additive_Done THEN
				State 			:= 1;
				Do_Cut 			:= FALSE;
				Done_Cut 		:= TRUE;
				S_Move_Velocity := FALSE;
				S_Move_Absolute := FALSE;
				S_Move_Additive := FALSE;
				S_Stop 			:= FALSE;
			END_IF

			IF Stop_Command OR Error_Command OR NOT Do_Cut THEN
				State 			:= 1;
				S_Move_Velocity := FALSE;
				S_Move_Absolute := FALSE;
				S_Move_Additive := FALSE;
				S_Stop 			:= FALSE;
			END_IF

		6: //Running in Manual Mode
			Power_Axis 		:= TRUE;
			Man_Mode_OFF 	:= FALSE;
			S_Move_Velocity := TRUE;
			S_Move_Additive := FALSE;
			S_Move_Absolute := FALSE;
			S_Stop 			:= FALSE;

			S_Velocity 		:= Blade_Pos;
			S_Direction 	:= 0;

			IF S_Velocity < 0 THEN
				S_Velocity 	:= -Blade_Pos;
				S_Direction := 1;
			END_IF
			IF Error_Command THEN
				State := 1;
			END_IF

			IF NOT Manual_Mode_Trigger THEN
				S_Move_Absolute_Done 	:= FALSE;
				State 					:= 7;
			END_IF

		7: //Sending Cutter Back to Original Position
			IF S_Actual_Position <> 0.0 THEN
				S_Velocity 		:= 50;
				S_Move_Velocity := FALSE;
				S_Move_Absolute := TRUE;
				S_Move_Additive := FALSE;
				S_Stop 			:= FALSE;
				S_Position 		:= 0.0;
				S_Direction 	:= 1;

				IF Error_Command THEN
					State := 1;
				END_IF
			END_IF
			IF S_Actual_Position = 0.0 THEN
				Man_Mode_OFF 	:= TRUE;
				State 			:= 1;
				Power_Axis 		:= FALSE;
				S_Move_Velocity := FALSE;
				S_Move_Absolute := FALSE;
				S_Move_Additive := FALSE;
				S_Stop 			:= FALSE;
			END_IF

			IF Error_Command THEN
				State := 1;
			END_IF

	END_CASE

	//Calling FSM_AXIS Function
	Slave(	Axis_Name 		:= ADR(gAxis02),
			Acceleration 	:= 5000,
			Deceleration 	:= 5000,
			Position 		:= S_Position,
			Distance 		:= S_Distance,
			Velocity 		:= S_Velocity,
			Direction 		:= S_Direction,
			Home 			:= Home_Axis,
			Power 			:= Power_Axis,
			Move_Velocity 	:= S_Move_Velocity,
			Move_Absolute 	:= S_Move_Absolute,
			Move_Additive 	:= S_Move_Additive,
			Stop 			:= S_Stop,
			Reset_Error 	:= Reset_Command);
	S_Active 				:= Slave.Active;
	S_Actual_Position 		:= Slave.Actual_Position;
	IF State = 3 OR State = 5 THEN
		S_Actual_Velocity := -Slave.Actual_Velocity;
	ELSE
		S_Actual_Velocity := Slave.Actual_Velocity;
	END_IF

	S_Move_Absolute_Done 	:= Slave.Move_Abs_Done;
	S_Move_Additive_Done 	:= Slave.Move_Add_Done;
	S_Homed 				:= Slave.Is_Homed;
	S_Powered 				:= Slave.Power_ON;
	S_Stoped 				:= Slave.Stop_Done;
	S_Error 				:= Slave.Error;

END_PROGRAM

PROGRAM _EXIT
	(* Insert code here *)

END_PROGRAM
```

### Program Logical/LED_IO (IEC)

#### Variables.var
```iecst
VAR
	State : INT := 0;
END_VAR
```

#### Main.st
```iecst
PROGRAM _INIT
	(* Insert code here *)

END_PROGRAM

PROGRAM _CYCLIC
	(* Insert code here *)
	(* Insert code here *)
	CASE State OF
		0: //Initiation
			DI1(LED_State := 'off');
			DI2(LED_State := 'off');
			DI3(LED_State := 'off');
			DI4(LED_State := 'off');
			DI5(LED_State := 'off');
			DI6(LED_State := 'off');

			IF M_Active AND Man_Mode_OFF THEN
				State := 2;
			END_IF

		1: //Error

			DI1(LED_State := 'off');
			DI2(LED_State := 'off');
			DI3(LED_State := 'off');
			DI4(LED_State := 'off');
			DI5(LED_State := 'off');
			DI6(LED_State := 'blink');

			Error_Command 	:= TRUE;
			Start_Command 	:= FALSE;
			Stop_Command 	:= TRUE;
			Power_Axis 		:= FALSE;

			IF Reset_Trigger AND Error_Trigger THEN
				Reset_Command 	:= TRUE;
				Error_Command 	:= FALSE;
			ELSIF Reset_Trigger AND NOT Error_Trigger THEN
				Reset_Command 	:= FALSE;
				Error_Command 	:= FALSE;
				State 			:= 2;
			END_IF

		2: //Disabled

			IF Error_Trigger THEN
				State 		:= 1;
			ELSIF Reset_Trigger THEN
				Power_Axis 	:= TRUE;
			END_IF

			DI1(LED_State := 'on');
			DI2(LED_State := 'on');
			DI3(LED_State := 'on');
			DI4(LED_State := 'on');
			DI5(LED_State := 'on');
			DI6(LED_State := 'on');

			IF M_Powered AND M_Homed THEN
				State := 4;
			ELSIF M_Powered AND NOT M_Homed THEN
				State := 3;
			END_IF
			IF NOT Man_Mode_OFF THEN
				State := 0;
			END_IF

		3: //Homing
			DI1(LED_State := 'blink');
			DI2(LED_State := 'blink');
			DI3(LED_State := 'blink');
			DI4(LED_State := 'blink');
			DI5(LED_State := 'blink');
			DI6(LED_State := 'blink');

			Home_Axis := TRUE;

			IF Error_Trigger THEN
				State 		:= 1;
			ELSIF M_Homed THEN
				Home_Axis 	:= FALSE;
				State 		:= 4;
			END_IF

			IF NOT Man_Mode_OFF THEN
				State := 0;
			END_IF

		4://Ready
			IF NOT (Conv_Lock_Trigger OR Conv_Lock_HMI_Trigger) THEN
				DI1(LED_State := 'off');
			END_IF
			IF NOT (Cutter_Lock_Trigger OR Cutter_Lock_HMI_Trigger) THEN
				DI2(LED_State := 'off');
			END_IF
			IF (Conv_Lock_Trigger OR Conv_Lock_HMI_Trigger) THEN
				DI1(LED_State := 'on');
			END_IF
			IF (Cutter_Lock_Trigger OR Cutter_Lock_HMI_Trigger) THEN
				DI2(LED_State := 'on');
			END_IF

			DI3(LED_State := 'blink');
			DI4(LED_State := 'off');
			DI5(LED_State := 'off');
			DI6(LED_State := 'off');

			Power_Axis := TRUE;

			IF Error_Trigger THEN
				State := 1;
			ELSIF Start_Trigger AND NOT Error_Trigger THEN
				State := 5;
			END_IF
			IF NOT Man_Mode_OFF THEN
				State := 0;
			END_IF

		5://Run
			IF NOT (Conv_Lock_Trigger OR Conv_Lock_HMI_Trigger) THEN
				DI1(LED_State := 'off');
			END_IF
			IF NOT (Cutter_Lock_Trigger OR Cutter_Lock_HMI_Trigger) THEN
				DI2(LED_State := 'off');
			END_IF
			IF (Conv_Lock_Trigger OR Conv_Lock_HMI_Trigger) THEN
				DI1(LED_State := 'on');
			END_IF
			IF (Cutter_Lock_Trigger OR Cutter_Lock_HMI_Trigger) THEN
				DI2(LED_State := 'on');
			END_IF

			DI3(LED_State := 'on');
			DI4(LED_State := 'on');
			DI5(LED_State := 'off');
			DI6(LED_State := 'off');

			Start_Command 	:= TRUE;
			Stop_Command 	:= FALSE;

			IF Error_Trigger THEN
				State := 1;
			ELSIF Sensor_Trigger THEN
				State := 8;
			ELSIF Stop_Trigger THEN
				Stop_Command 	:= TRUE;
				State 			:= 10;
			END_IF
			IF NOT Man_Mode_OFF THEN
				State := 0;
			END_IF

		8://Sensor Triggered
			IF NOT (Conv_Lock_Trigger OR Conv_Lock_HMI_Trigger) THEN
				DI1(LED_State := 'off');
			END_IF
			IF NOT (Cutter_Lock_Trigger OR Cutter_Lock_HMI_Trigger) THEN
				DI2(LED_State := 'off');
			END_IF
			IF (Conv_Lock_Trigger OR Conv_Lock_HMI_Trigger) THEN
				DI1(LED_State := 'on');
			END_IF
			IF (Cutter_Lock_Trigger OR Cutter_Lock_HMI_Trigger) THEN
				DI2(LED_State := 'on');
			END_IF

			DI3(LED_State := 'on');
			DI4(LED_State := 'on');
			DI5(LED_State := 'on');
			DI6(LED_State := 'off');

			IF Do_Cut THEN
				State := 9;
			ELSIF Stop_Trigger THEN
				Stop_Command 	:= TRUE;
				State 			:= 10;
			END_IF

			IF Error_Trigger THEN
				State := 1;
			END_IF

		9://Cutting in Operation
			IF NOT (Conv_Lock_Trigger OR Conv_Lock_HMI_Trigger) THEN
				DI1(LED_State := 'off');
			END_IF
			IF NOT (Cutter_Lock_Trigger OR Cutter_Lock_HMI_Trigger) THEN
				DI2(LED_State := 'off');
			END_IF
			IF (Conv_Lock_Trigger OR Conv_Lock_HMI_Trigger) THEN
				DI1(LED_State := 'on');
			END_IF
			IF (Cutter_Lock_Trigger OR Cutter_Lock_HMI_Trigger) THEN
				DI2(LED_State := 'on');
			END_IF

			DI3(LED_State := 'on');
			DI4(LED_State := 'on');
			DI5(LED_State := 'blink');
			DI6(LED_State := 'off');

			IF Done_Cut THEN
				State := 5;
			ELSIF Stop_Trigger THEN
				Stop_Command 	:= TRUE;
				State 			:= 10;
			END_IF

			IF Error_Trigger THEN
				State := 1;
			END_IF

		10://Stop

			Start_Command := FALSE;

			IF Error_Trigger THEN
				State := 1;
			ELSIF M_Stoped THEN
				State := 4;
			END_IF
			IF NOT Man_Mode_OFF THEN
				State := 0;
			END_IF

	END_CASE

END_PROGRAM

PROGRAM _EXIT
	(* Insert code here *)

END_PROGRAM
```

### Program Logical/Input_Bridge (IEC)

#### Main.st
```iecst
PROGRAM _INIT
	(* Insert code here *)
	//Initial Parameters

	Conv_Speed 		:= 100;
	Cut_Pos 		:= 50;
	Cutter_Speed 	:= 20;
	Cut_depth 		:= 50;

END_PROGRAM

PROGRAM _CYCLIC

	IF DiagCpuIsSimulated() THEN
		(* For Simulation *)
		//Operator
		//LED_IO Bridge
		Start_Trigger 			:= ComTCP_SimInputs.Start_Button_ButtonPress 		OR Start_Button_HMI;
		Stop_Trigger 			:= ComTCP_SimInputs.Stop_Button_ButtonPress 		OR Stop_Button_HMI;
		Error_Trigger 			:= ComTCP_SimInputs.Emergency_Button_ButtonToggle 	OR Emergancy_Button_HMI OR M_Error OR S_Error;
		Reset_Trigger 			:= ComTCP_SimInputs.White_Button_ButtonPress 		OR Reset_Button_HMI;
		Sensor_Trigger 			:= ComTCP_SimInputs.Yellow_Button_ButtonPress 		OR Sensor_Button_HMI;
		Conv_Lock_HMI_Trigger 	:= Conv_Lock_HMI;
		Cutter_Lock_HMI_Trigger := Cutter_Lock_HMI;

		IF Conv_Lock_HMI_Trigger THEN
			IF Conv_Speed_HMI < 10 THEN
				Conv_Speed 	:= 10;
			ELSE
				Conv_Speed 	:= Conv_Speed_HMI;
			END_IF
			IF Cutting_Pos_HMI < 10 THEN
				Cut_Pos 	:= 10;
			ELSE
				Cut_Pos 	:= Cutting_Pos_HMI;
			END_IF
		END_IF

		IF Cutter_Lock_HMI_Trigger THEN
			IF Cutter_Speed_HMI < 10 THEN
				Cutter_Speed 	:= 10;
			ELSE
				Cutter_Speed 	:= Cutter_Speed_HMI;
			END_IF
			IF Cutting_Depth_HMI < 10 THEN
				Cut_depth 		:= 10;
			ELSE
				Cut_depth 		:= Cutting_Depth_HMI;
			END_IF
		END_IF

		//Manual Motion
		Manual_Mode_Trigger := Man_Mode_HMI;
		Slow_Blade_Trigger 	:= Slow_Blade_HMI;
		Slow_Conv_Trigger 	:= Slow_Conv_HMI;
		IF Slow_Blade_Trigger THEN
			Blade_Pos := Blade_Man_HMI * 0.01 * 1000;
		ELSE
			Blade_Pos := Blade_Man_HMI * 1000;
		END_IF

		IF Slow_Conv_Trigger THEN
			Conv_Pos := Conv_Man_HMI * 0.01 *1000;
		ELSE
			Conv_Pos := Conv_Man_HMI * 1000;
		END_IF

	ELSE
		(* For Actual Setup *)
		Start_Trigger 			:= Start_Button OR Start_Button_HMI;
		Stop_Trigger 			:= Stop_Button OR Stop_Button_HMI;
		Error_Trigger 			:= Emergancy_Button_HMI OR M_Error OR S_Error;
		Reset_Trigger 			:= Reset_Button OR Reset_Button_HMI;
		Sensor_Trigger 			:= Sensor_Button OR Sensor_Button_HMI;
		Conv_Lock_HMI_Trigger 	:= Conv_Lock_HMI;
		Cutter_Lock_HMI_Trigger := Cutter_Lock_HMI;
		Conv_Lock_Trigger 		:= Conv_Lock;
		Cutter_Lock_Trigger 	:= Cutter_Lock;
		Over_Ride_Trigger 		:= Over_Ride_HMI;
		IF Over_Ride_Trigger THEN
			IF Conv_Lock_HMI_Trigger THEN
				IF Conv_Speed_HMI < 10 THEN
					Conv_Speed 	:= 10;
				ELSE
					Conv_Speed 	:= Conv_Speed_HMI;
				END_IF
				IF Cutting_Pos_HMI < 10 THEN
					Cut_Pos 	:= 10;
				ELSE
					Cut_Pos 	:= Cutting_Pos_HMI;
				END_IF
			END_IF
			IF Cutter_Lock_HMI_Trigger THEN
				IF Cutter_Speed_HMI < 10 THEN
					Cutter_Speed 	:= 10;
				ELSE
					Cutter_Speed 	:= Cutter_Speed_HMI;
				END_IF
				IF Cutting_Depth_HMI < 10 THEN
					Cut_depth 		:= 10;
				ELSE
					Cut_depth 		:= Cutting_Depth_HMI;
				END_IF
			END_IF
		ELSE
			IF Conv_Lock_Trigger AND NOT Cutter_Lock_Trigger THEN
				Conv_Speed 			:= (Speed*3000/32767);
				IF Speed < 10 THEN
					Conv_Speed 		:= 10;
				END_IF
				Cut_Pos 			:= (Position*1000/32767);
				IF Position < 10 THEN
					Cut_Pos 		:= 10;
				END_IF

			ELSIF Cutter_Lock_Trigger AND NOT Conv_Lock_Trigger THEN
				Cutter_Speed 		:= (Speed*3000/32767);
				IF Speed < 10 THEN
					Cutter_Speed 	:= 10;
				END_IF
				Cut_depth 			:= (Position*360/32767);
				IF Position < 10 THEN
					Cut_depth 		:= 10;
				END_IF
			ELSIF Conv_Lock_Trigger AND Cutter_Lock_Trigger THEN
				Error_Trigger 	:= TRUE;
			END_IF
		END_IF

		//Manual Motion
		Manual_Mode_Trigger := Man_Mode_HMI;
		Slow_Blade_Trigger 	:= Slow_Blade_HMI;
		Slow_Conv_Trigger 	:= Slow_Conv_HMI;
		IF Slow_Blade_Trigger THEN
			Blade_Pos 	:= Blade_Man_HMI * 0.01 * 1000;
		ELSE
			Blade_Pos 	:= Blade_Man_HMI*1000;
		END_IF

		IF Slow_Conv_Trigger THEN
			Conv_Pos 	:= Conv_Man_HMI * 0.01 * 1000;
		ELSE
			Conv_Pos 	:= Conv_Man_HMI*1000;
		END_IF
	END_IF

END_PROGRAM

PROGRAM _EXIT
	(* Insert code here *)

END_PROGRAM
```

### Program Logical/Output_Bridge (IEC)

#### Main.st
```iecst
PROGRAM _INIT
	(* Insert code here *)

END_PROGRAM

PROGRAM _CYCLIC
	(* Insert code here *)
	//Since when the motor not running it gives grabade values.
	IF NOT Start_Command THEN
		M_Actual_Velocity := 0;
		S_Actual_Velocity := 0;
	END_IF

	IF DiagCpuIsSimulated() THEN
		ComTCP_SimOutputs.Green_light_Key 	:= DI3.LED_Light;
		ComTCP_SimOutputs.Stop_light_Key 	:= DI4.LED_Light;
		ComTCP_SimOutputs.Yellow_light_Key 	:= DI5.LED_Light;
		ComTCP_SimOutputs.White_light_Key	:= DI6.LED_Light; //it will display red on real setup
		LED_DI1_HMI 						:= DI1.LED_Light;
		LED_DI2_HMI 						:= DI2.LED_Light;
		LED_DI3_HMI 						:= DI3.LED_Light;
		LED_DI4_HMI 						:= DI4.LED_Light;
		LED_DI5_HMI 						:= DI5.LED_Light;
		LED_DI6_HMI 						:= DI6.LED_Light;
		Dis_Conv_Speed_HMI 					:= M_Actual_Velocity/10;
		Dis_Cut_Speed_HMI 					:= S_Actual_Velocity/10;
		Dis_Cut_Pos_HMI 					:= REAL_TO_INT(Cut_Pos);
		Dis_Cut_Depth_HMI 					:= REAL_TO_INT(Cut_depth);

		//Master
		ComTCP_SimOutputs.Shaft_0_ACT_POS 	:= M_Actual_Position;

		//Slave
		ComTCP_SimOutputs.Shaft_1_ACT_POS 	:= S_Actual_Position;

	ELSE
		LED_DI1_HMI 		:= DI1.LED_Light;
		LED_DI2_HMI 		:= DI2.LED_Light;
		LED_DI3_HMI 		:= DI3.LED_Light;
		LED_DI4_HMI 		:= DI4.LED_Light;
		LED_DI5_HMI 		:= DI5.LED_Light;
		LED_DI6_HMI 		:= DI6.LED_Light;
		Dis_Conv_Speed_HMI 	:= M_Actual_Velocity/10;
		Dis_Cut_Speed_HMI 	:= S_Actual_Velocity/10;
		Dis_Cut_Pos_HMI 	:= REAL_TO_INT(Cut_Pos);
		Dis_Cut_Depth_HMI 	:= REAL_TO_INT(Cut_depth);

		//Hardware
		Display 			:= REAL_TO_INT((M_Actual_Velocity/10));

	END_IF

END_PROGRAM

PROGRAM _EXIT
	(* Insert code here *)

END_PROGRAM
```

Listed in the project but not available here: Logical/MNG_Global.typ, Logical/Global.typ, Logical/Libraries/ComTCP/ComTCP_P, Logical/acp10etxen, Logical/gAxis01obj/gAxis01a, Logical/gAxis02obj/gAxis02a, Logical/PLCopen, Logical/MyCamBis
